// TIA Portal V21 export
VAR_GLOBAL   // PLC tag table "K_Valvola_Filler"
END_VAR
VAR_GLOBAL CONSTANT   // user constants
   K_Valvola_Filler_IngressoProdotto : Int := 0;   // VA206
   K_Valvola_Filler_SicurezzaSprayBall : Int := 0;   // VA807
   K_Valvola_Filler_SprayallSerbatoioProdotto : Int := 0;   // VA801
   K_Valvola_Filler_LavaggioEsternoValvole : Int := 0;   // VA210
   K_Valvola_Filler_DrenaggioSerbatoioCIP : Int := 0;   // VA827
   K_Valvola_Filler_Rubinetti : Int := 0;   // EV NBNF
   K_Valvola_Filler_Vapore : Int := 0;
   K_Valvola_Filler_SlittaLavaggioPistoni : Int := 0;
   K_Valvola_Filler_IntercettoPompaCIP : Int := 0;   // VA817
   K_Valvola_Filler_BraccioLavaggioPistoni : Int := 0;
   K_Valvola_Filler_VaporeCip : Int := 0;
   K_Valvola_Filler_SoffioCameraPistoni : Int := 0;   // VA830
   K_Valvola_Filler_Sgolfatore : Int := 0;
   K_Valvola_Filler_LavaggioCameraPistoni : Int := 0;   // VA831
   K_Valvola_Filler_SoffioSensorePresenzaRiempitrice : Int := 0;   // VA03
   K_Valvola_Filler_VA214 : Int := 0;
   K_Valvola_Filler_VA215 : Int := 0;
   K_Valvola_Filler_VA220 : Int := 0;
   K_Valvola_Filler_FormazioneVuoto : Int := 0;   // VA229
   K_Valvola_Filler_AcquaPompaVuoto : Int := 0;   // VA230
   K_Valvola_Filler_DrenaggioSerbatoioVuoto : Int := 0;   // VA231
   K_Valvola_Filler_VA238 : Int := 0;
   K_Valvola_Filler_SvuotamentoTramoggiaConVuoto : Int := 0;   // VA265
   K_Valvola_Filler_LubrificazionePattino : Int := 0;   // VA233
   K_Valvola_Filler_IntercettoDaSerbVuotoASerbDrenaggio : Int := 0;   // VA256
   K_Valvola_Filler_SfiatoDaSerbVuotoASerbDrenaggio : Int := 0;
   K_Valvola_Filler_RipristinoVuotoSerbatoioDrenaggio : Int := 0;
   K_Valvola_Filler_VuotoDaNoCanNoFill : Int := 0;
   K_Valvola_Filler_VuotoPrimaParteRiempimento : Int := 0;   // VA260
   K_Valvola_Filler_DoppioVuoto : Int := 0;   // VA261
   K_Valvola_Filler_IntercettoPompaRiciclo : Int := 0;   // VA266
   K_Valvola_Filler_VA824 : Int := 0;
   K_Valvola_Filler_VA825 : Int := 0;
   K_Valvola_Filler_SprayballSerbatoioVuoto : Int := 0;   // VA850
   K_Valvola_Filler_VA851 : Int := 0;
   K_Valvola_Filler_LavaggioPistoniEstratti : Int := 0;   // VA263
   K_Valvola_Filler_IngressoSalamoiaSerbPreparazione : Int := 0;
   K_Valvola_Filler_IngressoOlioSerbPreparazione : Int := 0;
   K_Valvola_Filler_IntercettoVaporeSerbPreparazioneSalamoia : Int := 0;
   K_Valvola_Filler_IntercettoVaporeSerbPreparazioneOlio : Int := 0;
   K_Valvola_Filler_ModulanteVaporePreparazioneProdotto : Int := 0;
END_VAR
